FUNCTION_BLOCK DiagServer2 (* Sends sensor data and diagnostic data over a network. Wrapper for a SERVER function block. *)
  (* Standard: 61499-2; Description: A client can request measurements and diagnostic data from this function block. Requests should be made in regular intervals according to the data input DT. *)
  (* Version 1.0, 2017-08-27, Marc Jakobi, HTW Berlin *)
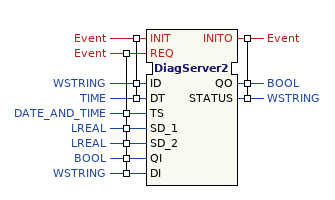
  EVENT_INPUT
    INIT WITH ID, DT; (* Initialization Request *)
    REQ WITH QI, SD_1, DI, SD_2, TS; (* Normal Execution Request *)
  END_EVENT
  EVENT_OUTPUT
    INITO WITH QO, STATUS; (* Initialization Confirm *)
  END_EVENT
  VAR_INPUT
    ID : WSTRING; (* Connection identifier *)
    DT : TIME := T#1m; (* Client request interval *)
    TS : DATE_AND_TIME; (* Time stamp *)
    SD_1 : LREAL; (* Input data *)
    SD_2 : LREAL; (* Input data *)
    QI : BOOL; (* Diagnostic qualifier *)
    DI : WSTRING; (* Diagnostic info *)
  END_VAR
  VAR_OUTPUT
    QO : BOOL; (* Output event qualifier *)
    STATUS : WSTRING; (* Service status *)
  END_VAR
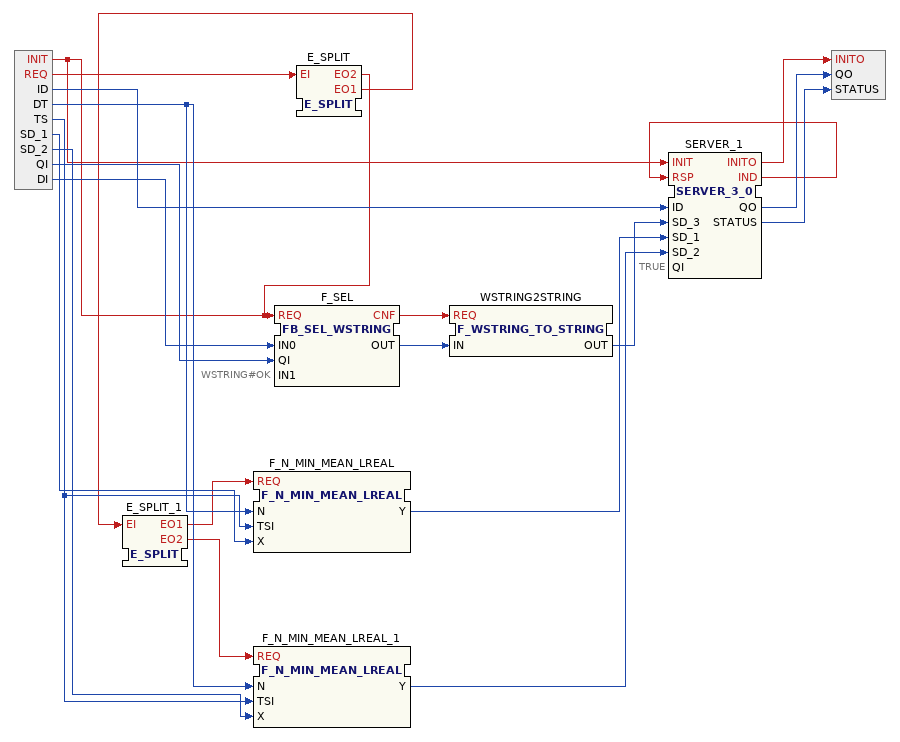
  FBS
    WSTRING2STRING : F_WSTRING_TO_STRING;
    SERVER_1 : SERVER_3_0(QI := TRUE);
    F_SEL : FB_SEL_WSTRING(IN1 := WSTRING#OK);
    E_SPLIT : E_SPLIT;
    F_N_MIN_MEAN_LREAL : F_N_MIN_MEAN_LREAL;
    F_N_MIN_MEAN_LREAL_1 : F_N_MIN_MEAN_LREAL;
    E_SPLIT_1 : E_SPLIT;
  END_FBS
  EVENT_CONNECTIONS
    INIT TO SERVER_1.INIT;
    SERVER_1.INITO TO INITO;
    INIT TO F_SEL.REQ;
    F_SEL.CNF TO WSTRING2STRING.REQ;
    REQ TO E_SPLIT.EI;
    E_SPLIT.EO2 TO F_SEL.REQ;
    SERVER_1.IND TO SERVER_1.RSP;
    E_SPLIT.EO1 TO E_SPLIT_1.EI;
    E_SPLIT_1.EO1 TO F_N_MIN_MEAN_LREAL.REQ;
    E_SPLIT_1.EO2 TO F_N_MIN_MEAN_LREAL_1.REQ;
  END_CONNECTIONS
  DATA_CONNECTIONS
    ID TO SERVER_1.ID;
    WSTRING2STRING.OUT TO SERVER_1.SD_3;
    SERVER_1.QO TO QO;
    SERVER_1.STATUS TO STATUS;
    DI TO F_SEL.IN0;
    F_SEL.OUT TO WSTRING2STRING.IN;
    QI TO F_SEL.QI;
    DT TO F_N_MIN_MEAN_LREAL.N;
    DT TO F_N_MIN_MEAN_LREAL_1.N;
    TS TO F_N_MIN_MEAN_LREAL.TSI;
    TS TO F_N_MIN_MEAN_LREAL_1.TSI;
    SD_1 TO F_N_MIN_MEAN_LREAL.X;
    SD_2 TO F_N_MIN_MEAN_LREAL_1.X;
    F_N_MIN_MEAN_LREAL.Y TO SERVER_1.SD_1;
    F_N_MIN_MEAN_LREAL_1.Y TO SERVER_1.SD_2;
  END_CONNECTIONS
END_FUNCTION_BLOCK
